PROGRAM myCounter
VAR
	
	iPumpCount AT %I* : UDINT;
	iGunRPMCount AT %I* : UDINT;
	iLastGunRPMCount : UDINT;
	
END_VAR

//plug both into EL1512 
//count chopper gun rpm (rising trigger)
	//add rpm hmi display (floating average)
IF iGunRPMCount <> iLastGunRPMCount THEN
	iLastGunRPMCount := iGunRPMCount;
END_IF
//count resin/mek pump strokes (rising trigger)
	//add flow rate hmi display (floating average)

END_PROGRAM

(* stored: Version 1.1.0.1, ProductVersion 3.1.4024.11
   POU myCounter: Id {426c8798-b4fe-4558-8c90-5e68c7e9353e}, SpecialFunc None *)
